{attribute addProperty BoxType "EK1100-0000-0018"}
{attribute addProperty Id "Beckhoff_EKM1xxxEK1122Beckhoff_EKM1xxxEK1122_7DC4CCD12586323.25"}
{attribute addProperty CRC "2798989831"}
{attribute addProperty SizeInBites "2586"}
{attribute addProperty SizeInBytes "323.25"}
TYPE Beckhoff_EKM1xxx_A6D53207 EXTENDS EK1100_179A0949 :
STRUCT
	{attribute addProperty Name "Beckhoff_EKM1xxxEK1122"}
	Beckhoff_EKM1xxxEK1122 : Beckhoff_EKM1xxxEK1122_7DC4CCD1;
END_STRUCT
END_TYPE

(* stored: Version 1.2.0.0, ProductVersion 3.1.4024.9
   DUT Beckhoff_EKM1xxx_A6D53207: Id {277dfbd4-a3b8-4873-b61e-2e8da240f620} *)
